PROGRAM Main_Algorithm
VAR
	module_executer: ARRAY[1..GVL_MODULES.n_modules] OF FB_Module_Executor;
	setup_inverter_comm: FB_Comm_Setup;
	setup_meter_comm: FB_Setup_Meter_Comm;
	i: UINT;
END_VAR

MAIN_1();
//MAIN_2();

METHOD MAIN_1 : BOOL
VAR_INPUT
END_VAR
VAR
	//load_from_db: LOAD_FROM_DB_FB;
END_VAR
IF GVL.WISNAM_PPC.START THEN			/// setup del simulatore ///
	setup_inverter_comm();
	setup_meter_comm();
	GVL.WISNAM_PPC.START := FALSE;
END_IF


module_executer[1](input := GVL_modules.read_meter);
module_executer[3](input := GVL_MODULES.acquire_setpoint_mqtt);
module_executer[4](input := GVL_modules.active_power_ctrl);
module_executer[5](input := GVL_modules.reactive_power_ctrl);
//IF NOT GVL_Freq.frequency_regulation_priority OR NOT GVL.WISNAM_PPC.actp_freq_reg_enabled THEN
//	module_executer[6](input := GVL_modules.command_dispatcher);
//END_IF
// load_from_db();
// test
END_METHOD

METHOD MAIN_2 : BOOL
VAR_INPUT
END_VAR
IF GVL.WISNAM_PPC.START THEN			/// setup del simulatore ///
	setup_inverter_comm();
	setup_meter_comm();
	GVL.WISNAM_PPC.START := FALSE;
END_IF


module_executer[1](input := GVL_modules.read_meter);
Update_Virtual_Meter();
module_executer[3](input := GVL_MODULES.acquire_setpoint_mqtt);
module_executer[4](input := GVL_modules.load_following);
module_executer[5](input := GVL_modules.reactive_power_ctrl);
module_executer[6](input := GVL_modules.command_dispatcher);
END_METHOD

METHOD MAIN_WIND_BESS : BOOL
VAR_INPUT
END_VAR
/// per tutte le funzioni "derivate" dal progetto originale Cosmo Eco, la potenza è espressa in termini assoluti e poi normalizzata qui ///
/// TO DO: valutare se mantenere questo approccio ///

/// Ciascuna delle funzioni richiamate restituisce variabili di tipo COMMAND SET (CMD_SET) 
/// TO DO: definire (lato progettazione) come devono essere ripartiti questi comandi e da quali moduli
/// Tutti questi moduli devono essere ridisegnati in fase di progettazione per l'interfacciamento con un sistema reale
END_METHOD

END_PROGRAM

(* stored: Version 1.1.0.1, ProductVersion 3.1.4026.11
   POU Main_Algorithm: Id {806268a4-dde8-408d-934c-2136314cd117}, SpecialFunc None
   Method MAIN_1: Id {bbcb920d-026a-4ea4-947e-2d8382fb6e38}
   Method MAIN_2: Id {9b3eb3c2-1e38-4d35-810f-949f998f5302}
   Method MAIN_WIND_BESS: Id {64f642b9-5327-4a67-9e64-752feb21fc07} *)
